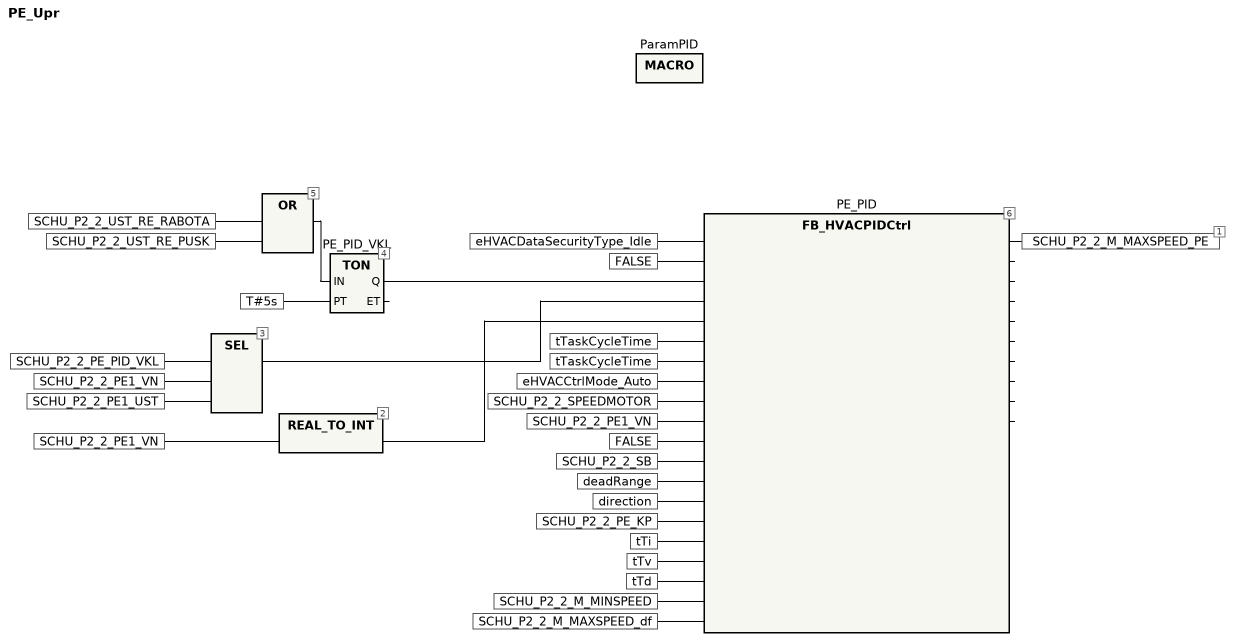
[picture p408: PE_Upr (CFC)]
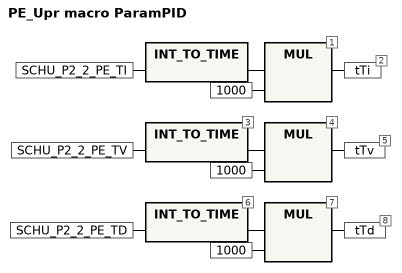
_CFC_ (* Continuous Function Chart, elements in execution order *)
#0 MACRO ParamPID()
	#1 INT_TO_TIME(SCHU_P2_2_PE_TI)
	#2 MUL(#1, 1000)
	#3 tTi <= #2
	#4 INT_TO_TIME(SCHU_P2_2_PE_TV)
	#5 MUL(#4, 1000)
	#6 tTv <= #5
	#7 INT_TO_TIME(SCHU_P2_2_PE_TD)
	#8 MUL(#7, 1000)
	#9 tTd <= #8
END_MACRO
#10 SCHU_P2_2_M_MAXSPEED_PE <= #15.out 1
#11 REAL_TO_INT(SCHU_P2_2_PE1_VN)
#12 SEL(SCHU_P2_2_PE_PID_VKL, SCHU_P2_2_PE1_VN, SCHU_P2_2_PE1_UST)
#13 PE_PID_VKL:TON(IN: #14, PT: T#5s)
#14 OR(SCHU_P2_2_UST_RE_RABOTA, SCHU_P2_2_UST_RE_PUSK)
#15 PE_PID:FB_HVACPIDCtrl(eHVACDataSecurityType_Idle, FALSE, #13.Q, #12, #11, tTaskCycleTime, tTaskCycleTime, eHVACCtrlMode_Auto, SCHU_P2_2_SPEEDMOTOR, SCHU_P2_2_PE1_VN, FALSE, SCHU_P2_2_SB, deadRange, direction, SCHU_P2_2_PE_KP, tTi, tTv, tTd, SCHU_P2_2_M_MINSPEED, SCHU_P2_2_M_MAXSPEED_df)
_END_CFC_
END_PROGRAM

(* POU IM/CHASTOTA_M1_M2, CFC *)
PROGRAM CHASTOTA_M1_M2
VAR
	RR: RAMP_REAL;
	SR_START_STER_REG: SR;
	SR_START_POV_REG: RS;
	RT_KOMVKL: R_TRIG;
	RT_KOMVKL_2: R_TRIG;
	RT_KOMVKL_1: R_TRIG;
	Zad_PE: TON;
END_VAR
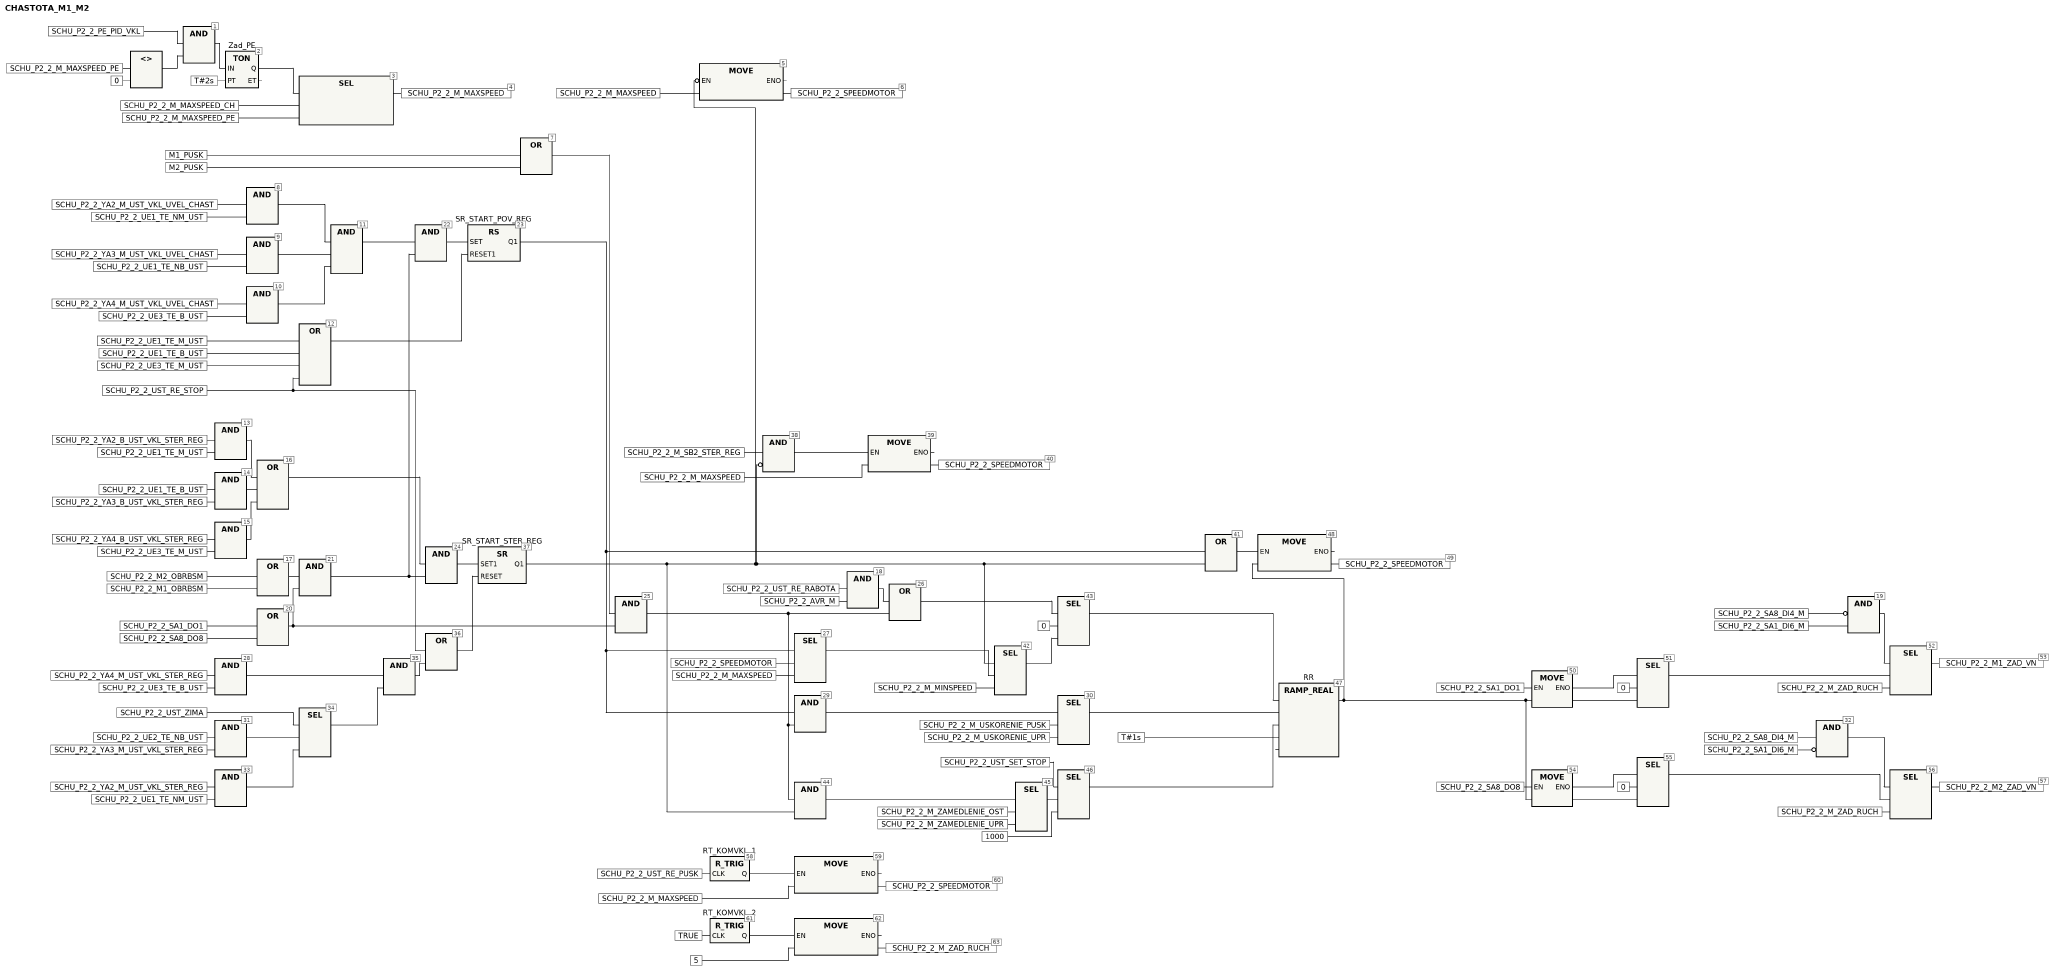
